// TIA Portal V21 export
VAR_GLOBAL   // PLC tag table "Default tag table"
   Start_SCL AT %I0.0 : Bool;
   Stop_SCL AT %I0.1 : Bool;
   Run_SCL AT %M0.0 : Bool;
   Start_LAD AT %I1.0 : Bool;
   Stop_LAD AT %I1.1 : Bool;
   Run_LAD AT %I1.2 : Bool;
END_VAR
